REGION Network 54: IS_SEOC ALARMS
   RUNG wire#powerrail
      Contact( "M_ONE" )
      wire#w1
      I_Contact( "DB16000_OPC_UA_TRIGGER_ALARM".CLIENT.U2_STA3_MEAS.ALARMS.MEAS_NOOZLE_CONNECTION_A )
      I_Contact( "DB16000_OPC_UA_TRIGGER_ALARM".CLIENT.U2_STA3_MEAS.ALARMS.MEAS_NOOZLE_METHOD_WORKING_BLOCKED_A )
      I_Contact( "DB16000_OPC_UA_TRIGGER_ALARM".CLIENT.U2_STA3_MEAS.ALARMS.MEAS_START_LAYER_CONNECTION_A )
      I_Contact( "DB16000_OPC_UA_TRIGGER_ALARM".CLIENT.U2_STA3_MEAS.ALARMS.MEAS_START_LAYER_METHOD_WORKING_BLOCKED_A )
      I_Contact( "DB16000_OPC_UA_TRIGGER_ALARM".CLIENT.U2_STA3_MEAS.ALARMS.MEAS_STOP_LAYER_CONNECTION_A )
      I_Contact( "DB16000_OPC_UA_TRIGGER_ALARM".CLIENT.U2_STA3_MEAS.ALARMS.MEAS_STOP_LAYER_METHOD_WORKING_BLOCKED_A )
      I_Contact( "DB16000_OPC_UA_TRIGGER_ALARM".CLIENT.U2_STA3_MEAS.ALARMS.CALIBRATE_CONNECTION_A )
      I_Contact( "DB16000_OPC_UA_TRIGGER_ALARM".CLIENT.U2_STA3_MEAS.ALARMS.CALIBRATE_METHOD_WORKING_BLOCKED_A )
      I_Contact( "DB16000_OPC_UA_TRIGGER_ALARM".CLIENT.U2_STA3_MEAS.ALARMS.RESET_CONNECTION_A )
      I_Contact( "DB16000_OPC_UA_TRIGGER_ALARM".CLIENT.U2_STA3_MEAS.ALARMS.RESET_METHOD_WORKING_BLOCKED_A )
      I_Contact( "DB16000_OPC_UA_TRIGGER_ALARM".CLIENT.U2_STA3_MEAS.ALARMS.READ_VAR_CONNECTION_A )
      I_Contact( "DB16000_OPC_UA_TRIGGER_ALARM".CLIENT.U2_STA3_MEAS.ALARMS.READ_VAR_METHOD_WORKING_BLOCKED_A )
      Not()
      Coil( #ALARM_AUX )
   END_RUNG
   RUNG wire#w1
      I_Contact( #ALARM_AUX )
      I_Contact( "DB16000_OPC_UA_TRIGGER_ALARM".CLIENT.U2_STA3_MEAS.ALARMS.PROFILER_CONFIG_A )
      I_Contact( "DB16000_OPC_UA_TRIGGER_ALARM".CLIENT.U2_STA3_MEAS.ALARMS.ANALYZER_CONFIG_A )
      I_Contact( "DB16000_OPC_UA_TRIGGER_ALARM".CLIENT.U2_STA3_MEAS.ALARMS.DMC_STRUCTURE_A )
      I_Contact( "DB16000_OPC_UA_TRIGGER_ALARM".CLIENT.U2_STA3_MEAS.ALARMS.ACQUISITION_A )
      I_Contact( "DB16000_OPC_UA_TRIGGER_ALARM".CLIENT.U2_STA3_MEAS.ALARMS.PROFILER_INIT_A )
      I_Contact( "DB16000_OPC_UA_TRIGGER_ALARM".CLIENT.U2_STA3_MEAS.ALARMS.DISTANCE_CALCULATION_A )
      I_Contact( "DB16000_OPC_UA_TRIGGER_ALARM".CLIENT.U2_STA3_MEAS.ALARMS.LAYER_GROWTH_A )
      I_Contact( "DB16000_OPC_UA_TRIGGER_ALARM".CLIENT.U2_STA3_MEAS.ALARMS.STORAGE_A )
      I_Contact( "DB16000_OPC_UA_TRIGGER_ALARM".CLIENT.U2_STA3_MEAS.ALARMS.DATABASE_CONNECTION_A )
      I_Contact( "DB16000_OPC_UA_TRIGGER_ALARM".CLIENT.U2_STA3_MEAS.ALARMS.CALIBRATION_MISSING_FIX_1_A )
      I_Contact( "DB16000_OPC_UA_TRIGGER_ALARM".CLIENT.U2_STA3_MEAS.ALARMS.CALIBRATION_MISSING_FIX_2_A )
      I_Contact( "DB16000_OPC_UA_TRIGGER_ALARM".CLIENT.U2_STA3_MEAS.ALARMS.CALIBRATION_MISSING_FIX_3_A )
      I_Contact( "DB16000_OPC_UA_TRIGGER_ALARM".CLIENT.U2_STA3_MEAS.ALARMS.CALIBRATION_MISSING_FIX_4_A )
      I_Contact( "DB16000_OPC_UA_TRIGGER_ALARM".CLIENT.U2_STA3_MEAS.ALARMS.CALIBRATION_PROC_A )
      I_Contact( "DB16000_OPC_UA_TRIGGER_ALARM".CLIENT.U2_STA3_MEAS.ALARMS.MEAS_NOOZLE_DISTANCE_ALARM )
      Not()
      Coil( #ALARM_AUX )
   END_RUNG
   RUNG wire#w1
      I_Contact( #ALARM_AUX )
      I_Contact( "DB16000_OPC_UA_TRIGGER_ALARM".CLIENT.U2_STA3_MEAS.ALARMS.CALIBRATION_OUT_RANGE_FIX_1_A )
      I_Contact( "DB16000_OPC_UA_TRIGGER_ALARM".CLIENT.U2_STA3_MEAS.ALARMS.CALIBRATION_OUT_RANGE_FIX_2_A )
      I_Contact( "DB16000_OPC_UA_TRIGGER_ALARM".CLIENT.U2_STA3_MEAS.ALARMS.CALIBRATION_OUT_RANGE_FIX_3_A )
      I_Contact( "DB16000_OPC_UA_TRIGGER_ALARM".CLIENT.U2_STA3_MEAS.ALARMS.CALIBRATION_OUT_RANGE_FIX_4_A )
      I_Contact( "DB16000_OPC_UA_TRIGGER_ALARM".CLIENT.U2_STA3_MEAS.ALARMS.PLC_PC_MAJOR_VERSIONS_MISMATCH_A )
      Not()
      Move(in := 16014, out1 => "DB440_MACHINE_ALARM_DECODING".GLOBAL_ALARMS_MACHINE.ALARM_DECODING)
      S_Coil( "DB440_MACHINE_ALARM_DECODING".ALARMS_UNIT_02.ST3_CLADDING.IS_SEOC_ALARMS )
   END_RUNG
   // the same network as SCL:
   #ALARM_AUX := NOT ("M_ONE" AND NOT "DB16000_OPC_UA_TRIGGER_ALARM".CLIENT.U2_STA3_MEAS.ALARMS.MEAS_NOOZLE_CONNECTION_A AND NOT "DB16000_OPC_UA_TRIGGER_ALARM".CLIENT.U2_STA3_MEAS.ALARMS.MEAS_NOOZLE_METHOD_WORKING_BLOCKED_A AND NOT "DB16000_OPC_UA_TRIGGER_ALARM".CLIENT.U2_STA3_MEAS.ALARMS.MEAS_START_LAYER_CONNECTION_A AND NOT "DB16000_OPC_UA_TRIGGER_ALARM".CLIENT.U2_STA3_MEAS.ALARMS.MEAS_START_LAYER_METHOD_WORKING_BLOCKED_A AND NOT "DB16000_OPC_UA_TRIGGER_ALARM".CLIENT.U2_STA3_MEAS.ALARMS.MEAS_STOP_LAYER_CONNECTION_A AND NOT "DB16000_OPC_UA_TRIGGER_ALARM".CLIENT.U2_STA3_MEAS.ALARMS.MEAS_STOP_LAYER_METHOD_WORKING_BLOCKED_A AND NOT "DB16000_OPC_UA_TRIGGER_ALARM".CLIENT.U2_STA3_MEAS.ALARMS.CALIBRATE_CONNECTION_A AND NOT "DB16000_OPC_UA_TRIGGER_ALARM".CLIENT.U2_STA3_MEAS.ALARMS.CALIBRATE_METHOD_WORKING_BLOCKED_A AND NOT "DB16000_OPC_UA_TRIGGER_ALARM".CLIENT.U2_STA3_MEAS.ALARMS.RESET_CONNECTION_A AND NOT "DB16000_OPC_UA_TRIGGER_ALARM".CLIENT.U2_STA3_MEAS.ALARMS.RESET_METHOD_WORKING_BLOCKED_A AND NOT "DB16000_OPC_UA_TRIGGER_ALARM".CLIENT.U2_STA3_MEAS.ALARMS.READ_VAR_CONNECTION_A AND NOT "DB16000_OPC_UA_TRIGGER_ALARM".CLIENT.U2_STA3_MEAS.ALARMS.READ_VAR_METHOD_WORKING_BLOCKED_A);
   #ALARM_AUX := NOT ("M_ONE" AND NOT #ALARM_AUX AND NOT "DB16000_OPC_UA_TRIGGER_ALARM".CLIENT.U2_STA3_MEAS.ALARMS.PROFILER_CONFIG_A AND NOT "DB16000_OPC_UA_TRIGGER_ALARM".CLIENT.U2_STA3_MEAS.ALARMS.ANALYZER_CONFIG_A AND NOT "DB16000_OPC_UA_TRIGGER_ALARM".CLIENT.U2_STA3_MEAS.ALARMS.DMC_STRUCTURE_A AND NOT "DB16000_OPC_UA_TRIGGER_ALARM".CLIENT.U2_STA3_MEAS.ALARMS.ACQUISITION_A AND NOT "DB16000_OPC_UA_TRIGGER_ALARM".CLIENT.U2_STA3_MEAS.ALARMS.PROFILER_INIT_A AND NOT "DB16000_OPC_UA_TRIGGER_ALARM".CLIENT.U2_STA3_MEAS.ALARMS.DISTANCE_CALCULATION_A AND NOT "DB16000_OPC_UA_TRIGGER_ALARM".CLIENT.U2_STA3_MEAS.ALARMS.LAYER_GROWTH_A AND NOT "DB16000_OPC_UA_TRIGGER_ALARM".CLIENT.U2_STA3_MEAS.ALARMS.STORAGE_A AND NOT "DB16000_OPC_UA_TRIGGER_ALARM".CLIENT.U2_STA3_MEAS.ALARMS.DATABASE_CONNECTION_A AND NOT "DB16000_OPC_UA_TRIGGER_ALARM".CLIENT.U2_STA3_MEAS.ALARMS.CALIBRATION_MISSING_FIX_1_A AND NOT "DB16000_OPC_UA_TRIGGER_ALARM".CLIENT.U2_STA3_MEAS.ALARMS.CALIBRATION_MISSING_FIX_2_A AND NOT "DB16000_OPC_UA_TRIGGER_ALARM".CLIENT.U2_STA3_MEAS.ALARMS.CALIBRATION_MISSING_FIX_3_A AND NOT "DB16000_OPC_UA_TRIGGER_ALARM".CLIENT.U2_STA3_MEAS.ALARMS.CALIBRATION_MISSING_FIX_4_A AND NOT "DB16000_OPC_UA_TRIGGER_ALARM".CLIENT.U2_STA3_MEAS.ALARMS.CALIBRATION_PROC_A AND NOT "DB16000_OPC_UA_TRIGGER_ALARM".CLIENT.U2_STA3_MEAS.ALARMS.MEAS_NOOZLE_DISTANCE_ALARM);
   IF NOT ("M_ONE" AND NOT #ALARM_AUX AND NOT "DB16000_OPC_UA_TRIGGER_ALARM".CLIENT.U2_STA3_MEAS.ALARMS.CALIBRATION_OUT_RANGE_FIX_1_A AND NOT "DB16000_OPC_UA_TRIGGER_ALARM".CLIENT.U2_STA3_MEAS.ALARMS.CALIBRATION_OUT_RANGE_FIX_2_A AND NOT "DB16000_OPC_UA_TRIGGER_ALARM".CLIENT.U2_STA3_MEAS.ALARMS.CALIBRATION_OUT_RANGE_FIX_3_A AND NOT "DB16000_OPC_UA_TRIGGER_ALARM".CLIENT.U2_STA3_MEAS.ALARMS.CALIBRATION_OUT_RANGE_FIX_4_A AND NOT "DB16000_OPC_UA_TRIGGER_ALARM".CLIENT.U2_STA3_MEAS.ALARMS.PLC_PC_MAJOR_VERSIONS_MISMATCH_A) THEN
       "DB440_MACHINE_ALARM_DECODING".GLOBAL_ALARMS_MACHINE.ALARM_DECODING := 16014;
       "DB440_MACHINE_ALARM_DECODING".ALARMS_UNIT_02.ST3_CLADDING.IS_SEOC_ALARMS := TRUE;
   END_IF;
END_REGION

REGION Network 55: WARNINGS
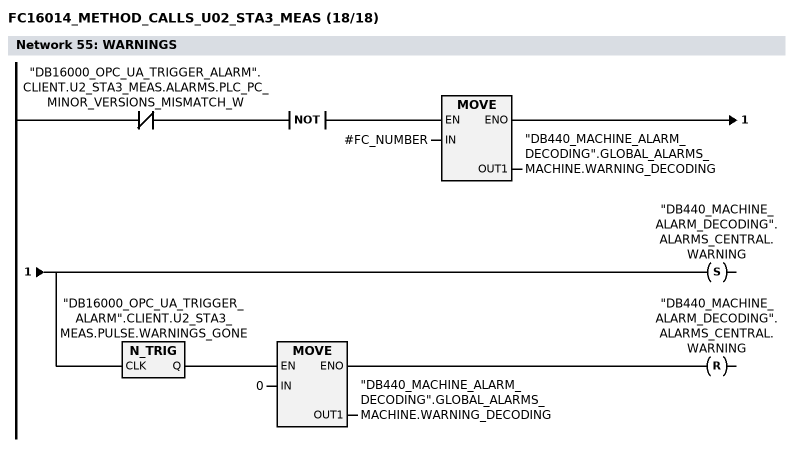
   RUNG wire#powerrail
      I_Contact( "DB16000_OPC_UA_TRIGGER_ALARM".CLIENT.U2_STA3_MEAS.ALARMS.PLC_PC_MINOR_VERSIONS_MISMATCH_W )
      Not()
      Move(in := #FC_NUMBER, out1 => "DB440_MACHINE_ALARM_DECODING".GLOBAL_ALARMS_MACHINE.WARNING_DECODING)
      wire#w1
      S_Coil( "DB440_MACHINE_ALARM_DECODING".ALARMS_CENTRAL.WARNING )
   END_RUNG
   RUNG wire#w1
      N_Trig( "DB16000_OPC_UA_TRIGGER_ALARM".CLIENT.U2_STA3_MEAS.PULSE.WARNINGS_GONE )
      Move(in := 0, out1 => "DB440_MACHINE_ALARM_DECODING".GLOBAL_ALARMS_MACHINE.WARNING_DECODING)
      R_Coil( "DB440_MACHINE_ALARM_DECODING".ALARMS_CENTRAL.WARNING )
   END_RUNG
   // the same network as SCL:
   #_w1 := NOT (NOT "DB16000_OPC_UA_TRIGGER_ALARM".CLIENT.U2_STA3_MEAS.ALARMS.PLC_PC_MINOR_VERSIONS_MISMATCH_W);
   IF #_w1 THEN
       "DB440_MACHINE_ALARM_DECODING".GLOBAL_ALARMS_MACHINE.WARNING_DECODING := #FC_NUMBER;
       "DB440_MACHINE_ALARM_DECODING".ALARMS_CENTRAL.WARNING := TRUE;
   END_IF;
   #_w2 := NOT #_w1 AND "DB16000_OPC_UA_TRIGGER_ALARM".CLIENT.U2_STA3_MEAS.PULSE.WARNINGS_GONE;   // falling edge
   "DB16000_OPC_UA_TRIGGER_ALARM".CLIENT.U2_STA3_MEAS.PULSE.WARNINGS_GONE := #_w1;
   IF #_w2 THEN
       "DB440_MACHINE_ALARM_DECODING".GLOBAL_ALARMS_MACHINE.WARNING_DECODING := 0;
       "DB440_MACHINE_ALARM_DECODING".ALARMS_CENTRAL.WARNING := FALSE;
   END_IF;
END_REGION
END_FUNCTION
